(* IEC 61131-3 sources: eCockpitGit/test_project/src/%F%00 Library/%F%Common Functions/%F%Linearsation/%F%WORD, 4 files *)

(* ---- %POU%FU_wLinear2.st ---- *)
//This function, converts an x, value to an y value using and 2 points on the x and y scale
// |**Version**|**Author**| **Date** |**Changes**
// | 1         | NSN      | 21-06-18 | Creation
// | 2         | NSN      | 24-05-22 | Fixed cases where y difference was negative
FUNCTION FU_wLinear2 : WORD
VAR_INPUT
	XIn		:WORD;
	X1		:WORD;
	X2		:WORD;
	Y1		:WORD;
	Y2		:WORD;
END_VAR
VAR
	a		:REAL;
	b		:REAL;
END_VAR
(*%!%__DELIMITER__%!%*)
IF X2 > X1 THEN
	//a value is calculated
	IF X2 - X1 = 0 THEN	a := 0; ELSE a := (TO_REAL(Y2) - TO_REAL(Y1)) / (TO_REAL(X2) - TO_REAL(X1)); END_IF
	//b value is calculated
	b 							:=		TO_REAL(Y1) - (a * TO_REAL(X1));
	//Output is calculated
	FU_wLinear2 				:=		TO_WORD(a * TO_REAL (XIn) + b);
ELSE
	//a value is calculated
	IF X2 - X1 = 0 THEN	a := 0; ELSE a := (TO_REAL(Y2) - TO_REAL(Y1)) / (TO_REAL(X2) - TO_REAL(X1)); END_IF
	//b value is calculated
	b 							:=		TO_REAL(Y1) - (a * TO_REAL(X1));
	//Output is calculated
	FU_wLinear2 				:=		TO_WORD(a * TO_REAL (XIn) + b);
END_IF

(* ---- %POU%FU_wLinear2Ends.st ---- *)
//This function, converts an x, value to an y value using and 2 points on the x and y scale
//This function has ends, which means the output is never greater or smaller than the range of y
// |**Version**|**Author**| **Date** |**Changes**
// | 1         | NSN      | 21-06-18 | Creation
// | 2         | NSN      | 24-05-22 | Fixed cases where y difference was negative
FUNCTION FU_wLinear2Ends : WORD
VAR_INPUT
	XIn		:WORD;
	X1		:WORD;
	X2		:WORD;
	Y1		:WORD;
	Y2		:WORD;
END_VAR
VAR
	a		:REAL;
	b		:REAL;
END_VAR
(*%!%__DELIMITER__%!%*)
IF X2 > X1 THEN
	IF XIn <= X1 THEN	//When input is out of bounds
		FU_wLinear2Ends 			:=		Y1;
	ELSIF XIn >= X2 THEN	//When input is out of bounds
		FU_wLinear2Ends 			:=		Y2;
	ELSIF XIn > X1 AND XIn < X2 THEN	//When input is with the
		//a value is calculated
		IF X2 - X1 = 0 THEN	a := 0; ELSE a := (TO_REAL(Y2) - TO_REAL(Y1)) / (TO_REAL(X2) - TO_REAL(X1)); END_IF
		//b value is calculated
		b 							:=		TO_REAL(Y1) - (a * TO_REAL(X1));
		//Output is calculated
		FU_wLinear2Ends 			:=		TO_WORD(a * TO_REAL (XIn) + b);
	END_IF
ELSE
	IF XIn >= X1 THEN
		FU_wLinear2Ends 			:=		Y1;
	ELSIF XIn <= X2 THEN
		FU_wLinear2Ends 			:=		Y2;
	ELSIF XIn < X1 AND XIn > X2 THEN
		//a value is calculated
		IF X2 - X1 = 0 THEN	a := 0; ELSE a := (TO_REAL(Y2) - TO_REAL(Y1)) / (TO_REAL(X2) - TO_REAL(X1)); END_IF
		//b value is calculated
		b 							:=		TO_REAL(Y1) - (a * TO_REAL(X1));
		//Output is calculated
		FU_wLinear2Ends 			:=		TO_WORD(a * TO_REAL (XIn) + b);
	END_IF
END_IF

(* ---- %POU%FU_wLinear3Ends.st ---- *)
//This function, converts an x, value to an y value using and 3 points on the x and y scale
//This function has ends, which means the output is never greater or smaller than the range of y
// |**Version**|**Author**| **Date** |**Changes**
// | 1         | NSN      | 10-01-18 | Updated to new format
// | 1.1       | NSN      | 13-06-18 | Updated names and types
// | 2         | NSN      | 24-05-22 | Fixed cases where y difference was negative
FUNCTION FU_wLinear3Ends : WORD
VAR_INPUT
	XIn		:WORD;
	X1		:WORD;
	X2		:WORD;
	X3		:WORD;
	Y1		:WORD;
	Y2		:WORD;
	Y3		:WORD;
END_VAR
VAR
	a		:REAL;
	b		:REAL;
END_VAR
(*%!%__DELIMITER__%!%*)
IF X3 > X1 THEN
	IF XIn <= X1 THEN	//When input is out of bounds
		FU_wLinear3Ends 			:=		Y1;
	ELSIF XIn >= X3 THEN	//When input is out of bounds
		FU_wLinear3Ends 			:=		Y3;
	ELSIF XIn > X1 AND XIn <= X2 THEN	//When input is with the
		//a value is calculated
		IF X2 - X1 = 0 THEN	a := 0; ELSE a := (TO_REAL(Y2) - TO_REAL(Y1)) / (TO_REAL(X2) - TO_REAL(X1)); END_IF
		//b value is calculated
		b 							:=		TO_REAL(Y1) - (a * TO_REAL(X1));
		//Output is calculated
		FU_wLinear3Ends 			:=		TO_WORD(a * TO_REAL (XIn) + b);
	ELSIF XIn > X2 AND XIn < X3 THEN
		//a value is calculated
		IF X3 - X2 = 0 THEN	a := 0; ELSE a := (TO_REAL(Y3) - TO_REAL(Y2)) / (TO_REAL(X3) - TO_REAL(X2)); END_IF
		//b value is calculated
		b 							:=		TO_REAL(Y2) - (a * TO_REAL(X2));
		//Output is calculated
		FU_wLinear3Ends 			:=		TO_WORD(a * TO_REAL (XIn) + b);
	END_IF
ELSE
	IF XIn >= X1 THEN
		FU_wLinear3Ends 			:=		Y1;
	ELSIF XIn <= X3 THEN
		FU_wLinear3Ends 			:=		Y3;
	ELSIF XIn < X1 AND XIn >= X2 THEN
		//a value is calculated
		IF X2 - X1 = 0 THEN	a := 0; ELSE a := (TO_REAL(Y2) - TO_REAL(Y1)) / (TO_REAL(X2) - TO_REAL(X1)); END_IF
		//b value is calculated
		b 							:=		TO_REAL(Y1) - (a * TO_REAL(X1));
		//Output is calculated
		FU_wLinear3Ends 			:=		TO_WORD(a * TO_REAL (XIn) + b);
	ELSIF XIn < X2 AND XIn > X3 THEN
		//a value is calculated
		IF X3 - X2 = 0 THEN	a := 0; ELSE a := (TO_REAL(Y3) - TO_REAL(Y2)) / (TO_REAL(X3) - TO_REAL(X2)); END_IF
		//b value is calculated
		b 							:=		TO_REAL(Y2) - (a * TO_REAL(X2));
		//Output is calculated
		FU_wLinear3Ends 			:=		TO_WORD(a * TO_REAL (XIn) + b);
	END_IF
END_IF

(* ---- %POU%FU_wLinear4Ends.st ---- *)
//This function, converts an x, value to an y value using and 3 points on the x and y scale
//This function has ends, which means the output is never greater or smaller than the range of y
// |**Version**|**Author**| **Date** |**Changes**
// | 1         | NSN      | 30-05-18 | Updated to new format
// | 2         | NSN      | 24-05-22 | Fixed cases where y difference was negative
FUNCTION FU_wLinear4Ends : WORD
VAR_INPUT
	XIn		:WORD;
	X1		:WORD;
	X2		:WORD;
	X3		:WORD;
	X4		:WORD;
	Y1		:WORD;
	Y2		:WORD;
	Y3		:WORD;
	Y4		:WORD;
END_VAR
VAR
	a		:REAL;
	b		:REAL;
END_VAR
(*%!%__DELIMITER__%!%*)
IF X4 > X1 THEN
	IF XIn <= X1 THEN	//When input is out of bounds
		FU_wLinear4Ends 			:=		Y1;
	ELSIF XIn >= X4 THEN	//When input is out of bounds
		FU_wLinear4Ends 			:=		Y4;
	ELSIF XIn > X1 AND XIn <= X2 THEN	//When input is with the
		//a value is calculated
		IF X2 - X1 = 0 THEN	a := 0; ELSE a := (TO_REAL(Y2) - TO_REAL(Y1)) / (TO_REAL(X2) - TO_REAL(X1)); END_IF
		//b value is calculated
		b 							:=		TO_REAL(Y1) - (a * TO_REAL(X1));
		//Output is calculated
		FU_wLinear4Ends 			:=		TO_WORD(a * TO_REAL (XIn) + b);
	ELSIF XIn > X2 AND XIn <= X3 THEN
		//a value is calculated
		IF X3 - X2 = 0 THEN	a := 0; ELSE a := (TO_REAL(Y3) - TO_REAL(Y2)) / (TO_REAL(X3) - TO_REAL(X2)); END_IF
		//b value is calculated
		b 							:=		TO_REAL(Y2) - (a * TO_REAL(X2));
		//Output is calculated
		FU_wLinear4Ends 			:=		TO_WORD(a * TO_REAL (XIn) + b);
	ELSIF XIn > X3 AND XIn < X4 THEN
		//a value is calculated
		IF X4 - X3 = 0 THEN	a := 0; ELSE a := (TO_REAL(Y4) - TO_REAL(Y3)) / (TO_REAL(X4) - TO_REAL(X3)); END_IF
		//b value is calculated
		b 							:=		TO_REAL(Y3) - (a * TO_REAL(X3));
		//Output is calculated
		FU_wLinear4Ends 			:=		TO_WORD(a * TO_REAL (XIn) + b);
	END_IF
ELSE
	IF XIn >= X1 THEN
		FU_wLinear4Ends 			:=		Y1;
	ELSIF XIn <= X4 THEN
		FU_wLinear4Ends 			:=		Y4;
	ELSIF XIn < X1 AND XIn >= X2 THEN
		//a value is calculated
		IF X2 - X1 = 0 THEN	a := 0; ELSE a := (TO_REAL(Y2) - TO_REAL(Y1)) / (TO_REAL(X2) - TO_REAL(X1)); END_IF
		//b value is calculated
		b 							:=		TO_REAL(Y1) - (a * TO_REAL(X1));
		//Output is calculated
		FU_wLinear4Ends 			:=		TO_WORD(a * TO_REAL (XIn) + b);
	ELSIF XIn < X2 AND XIn >= X3 THEN
		//a value is calculated
		IF X3 - X2 = 0 THEN	a := 0; ELSE a := (TO_REAL(Y3) - TO_REAL(Y2)) / (TO_REAL(X3) - TO_REAL(X2)); END_IF
		//b value is calculated
		b 							:=		TO_REAL(Y2) - (a * TO_REAL(X2));
		//Output is calculated
		FU_wLinear4Ends 			:=		TO_WORD(a * TO_REAL (XIn) + b);
	ELSIF XIn < X3 AND XIn > X4 THEN
		//a value is calculated
		IF X4 - X3 = 0 THEN	a := 0; ELSE a := (TO_REAL(Y4) - TO_REAL(Y3)) / (TO_REAL(X4) - TO_REAL(X3)); END_IF
		//b value is calculated
		b 							:=		TO_REAL(Y3) - (a * TO_REAL(X3));
		//Output is calculated
		FU_wLinear4Ends 			:=		TO_WORD(a * TO_REAL (XIn) + b);
	END_IF
END_IF
